INTERFACE I_AdjustablePump EXTENDS I_Pump, __SYSTEM.IQueryInterface

METHOD SetFlowRate : BOOL
VAR_INPUT
	fNewRate : REAL;
END_VAR
END_METHOD

END_INTERFACE

(* stored: Version 1.1.0.1, ProductVersion 3.1.4024.16
   Itf I_AdjustablePump: Id {148dce30-640d-4911-ac1d-63b30a1cb7ed}
   Method SetFlowRate: Id {e4e255d7-7992-44e2-aa39-b30bb0c1a410} *)
